// Mitsubishi GX Works2 project: rez_big_sizes   PLC: FX3G

// global labels: Global1
VAR_GLOBAL CONSTANT
  fot : BOOL;
END_VAR

PROGRAM MAIN
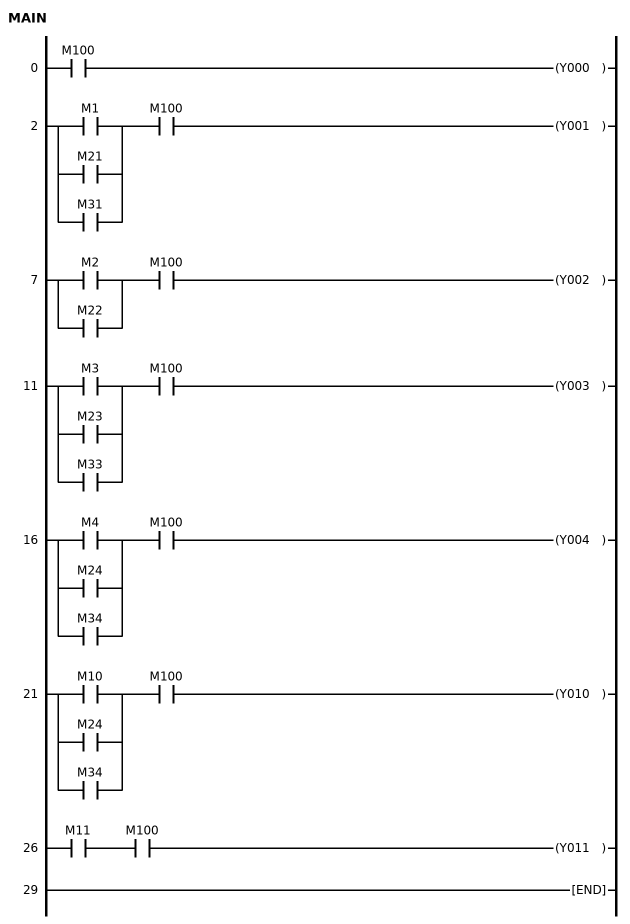
0     LD      M100
      OUT     Y000
2     LD      M1
      OR      M21
      OR      M31
      AND     M100
      OUT     Y001
7     LD      M2
      OR      M22
      AND     M100
      OUT     Y002
11    LD      M3
      OR      M23
      OR      M33
      AND     M100
      OUT     Y003
16    LD      M4
      OR      M24
      OR      M34
      AND     M100
      OUT     Y004
21    LD      M10
      OR      M24
      OR      M34
      AND     M100
      OUT     Y010
26    LD      M11
      AND     M100
      OUT     Y011
29    END
END_PROGRAM

PROGRAM panel
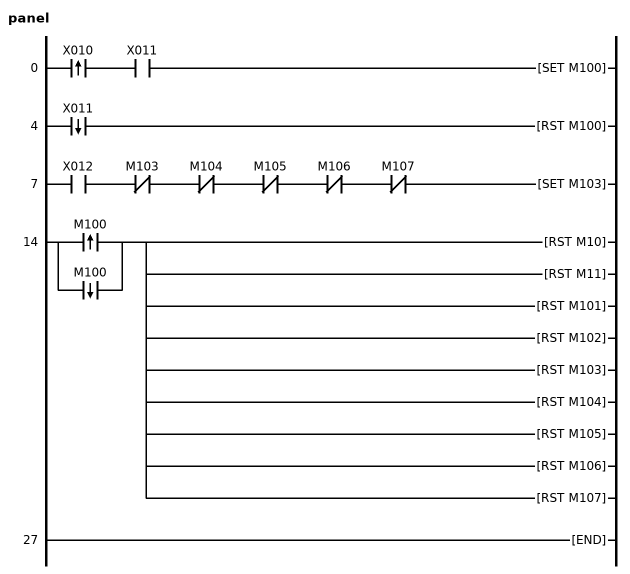
0     LDP     X010
      AND     X011
      SET     M100
4     LDF     X011
      RST     M100
7     LD      X012
      ANI     M103
      ANI     M104
      ANI     M105
      ANI     M106
      ANI     M107
      SET     M103
14    LDP     M100
      ORF     M100
      RST     M10
      RST     M11
      RST     M101
      RST     M102
      RST     M103
      RST     M104
      RST     M105
      RST     M106
      RST     M107
27    END
END_PROGRAM

PROGRAM size_sel
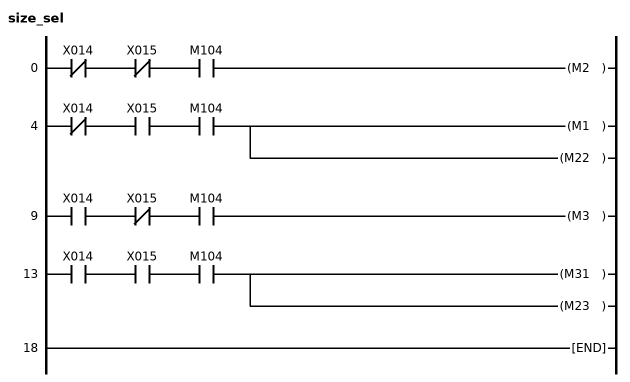
0     LDI     X014
      ANI     X015
      AND     M104
      OUT     M2
4     LDI     X014
      AND     X015
      AND     M104
      OUT     M1
      OUT     M22
9     LD      X014
      ANI     X015
      AND     M104
      OUT     M3
13    LD      X014
      AND     X015
      AND     M104
      OUT     M31
      OUT     M23
18    END
END_PROGRAM

PROGRAM work_st
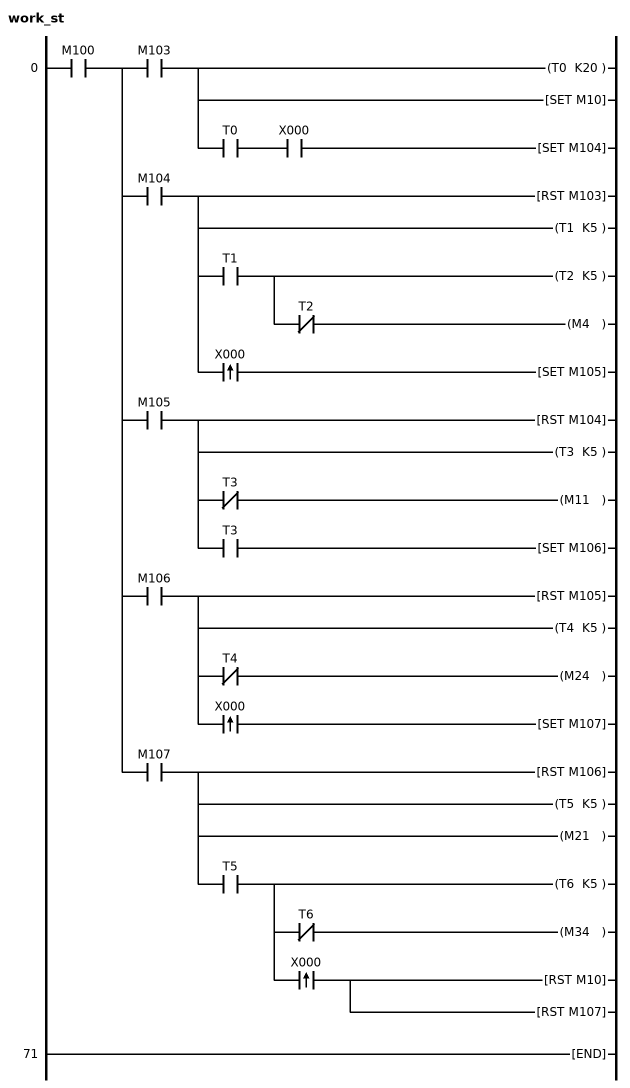
0     LD      M100
      MPS
      AND     M103
      OUT     T0 K20
      SET     M10
      AND     T0
      AND     X000
      SET     M104
      MRD
      AND     M104
      RST     M103
      OUT     T1 K5
      MPS
      AND     T1
      OUT     T2 K5
      ANI     T2
      OUT     M4
      MPP
      ANDP    X000
      SET     M105
      MRD
      AND     M105
      RST     M104
      OUT     T3 K5
      MPS
      ANI     T3
      OUT     M11
      MPP
      AND     T3
      SET     M106
      MRD
      AND     M106
      RST     M105
      OUT     T4 K5
      MPS
      ANI     T4
      OUT     M24
      MPP
      ANDP    X000
      SET     M107
      MPP
      AND     M107
      RST     M106
      OUT     T5 K5
      OUT     M21
      AND     T5
      OUT     T6 K5
      MPS
      ANI     T6
      OUT     M34
      MPP
      ANDP    X000
      RST     M10
      RST     M107
71    END
END_PROGRAM
